// TIA Portal V18 export
FUNCTION_BLOCK "FB_Next"   // FB42, SCL
{ S7_Optimized_Access := 'TRUE' }
AUTHOR : Sachs
FAMILY : General
VERSION : 1.0
// stored: AutoNumber true, IsIECCheckEnabled false, IsRetainMemResEnabled false, MemoryReserve 100, SetENOAutomatically false, UDAEnableTagReadback false
   VAR_INPUT
      I_bEnable : Bool;
      I_bSeqMode : Bool;
      I_tTimeValue : Time;
   END_VAR
   VAR_OUTPUT
      O_bStart : Bool;
   END_VAR
   VAR
      ton_Delay { S7_SetPoint := 'True'} : TON_TIME;
      bStartdelay : Bool;
   END_VAR
BEGIN
   //***********************************************************************************************
   //Function:
   //
   //Additional Blocks & Libraries:
   //  None
   //  
   //Version   Date        Person  Description
   //1.0       04.11.15    Sachs   Creation
   //1.0       15.03.2016  Sachs   
   //***********************************************************************************************

   //***********************************************************************************************
   //下一步跳转模块/next step
   //***********************************************************************************************
   //延时条件
   IF #I_bEnable AND #I_bSeqMode AND (#ton_Delay.Q = FALSE OR #I_tTimeValue = t#0s) THEN
       #bStartdelay := TRUE;    
   END_IF;

   #ton_Delay(IN := #bStartdelay,
              PT := #I_tTimeValue);

   #O_bStart := #ton_Delay.Q;

   IF #ton_Delay.Q OR NOT #I_bEnable THEN
       #bStartdelay := FALSE; 
   END_IF;
END_FUNCTION_BLOCK
